FUNCTION_BLOCK FB_Wirefabricator EXTENDS FB_StoneFurnace IMPLEMENTS I_2InputConversion
VAR
	test: int;
END_VAR

tProductionTime := T#0.5S;
test :=2;
SUPER^();

{error 'add property implementation or delete property to use base implementation'}
PROPERTY ProductsOut : UINT
GET
END_GET
END_PROPERTY

END_FUNCTION_BLOCK

(* stored: Version 1.1.0.1, ProductVersion 3.1.4026.8
   POU FB_Wirefabricator: Id {5876c030-de8a-45f1-8f9e-e7f8eb8e019f}, SpecialFunc None
   Property ProductsOut: Id {06e8bf58-1955-493c-8791-796cb3ec5297}
   Get Get: Id {bd177913-e17e-4ff5-9554-89466941e9c9} *)
